// TIA Portal V17 export
// export: Created 2023-02-25T14:39:28.1459249Z, ExportSetting WithDefaults, DisplayName Totally Integrated Automation Portal, DisplayVersion V17, DisplayName TIA Portal Openness, DisplayVersion V17, DisplayName TIA Portal Version Control Interface, DisplayVersion V17, DisplayName TIA Portal Test Suite Advanced, DisplayVersion V17, DisplayName STEP 7 Professional, DisplayVersion V17, DisplayName SIMATIC Energy Suite, DisplayVersion V17, DisplayName STEP 7 Safety, DisplayVersion V17, DisplayName WinCC Professional, DisplayVersion V17
FUNCTION_BLOCK "HW_MotorControle"   // FB1, LAD
{ S7_Optimized_Access := 'TRUE' }
VERSION : 0.1
// stored: AutoNumber true, IsIECCheckEnabled false, IsRetainMemResEnabled false, MemoryReserve 100, SetENOAutomatically false, UDAEnableTagReadback false
   VAR_INPUT
      inConveyor : "stt_Motor";
      FirstScan : Bool;
   END_VAR
   VAR_OUTPUT
      Conveyor : Real;
   END_VAR
   VAR
      S1 : Bool;
      S2 : Bool;
      S3 : Bool;
      S4 : Bool;
      S5 : Bool;
      t1 : Bool;
      t2 : Bool;
      speedLeft : Real;
      IEC_Timer_0_Instance { ExternalAccessible := 'False'; ExternalVisible := 'False'; ExternalWritable := 'False'} : TON_TIME;
      IEC_Timer_0_Instance_1 { ExternalAccessible := 'False'; ExternalVisible := 'False'; ExternalWritable := 'False'} : TON_TIME;
   END_VAR
BEGIN

REGION Network 1: Step 2-1
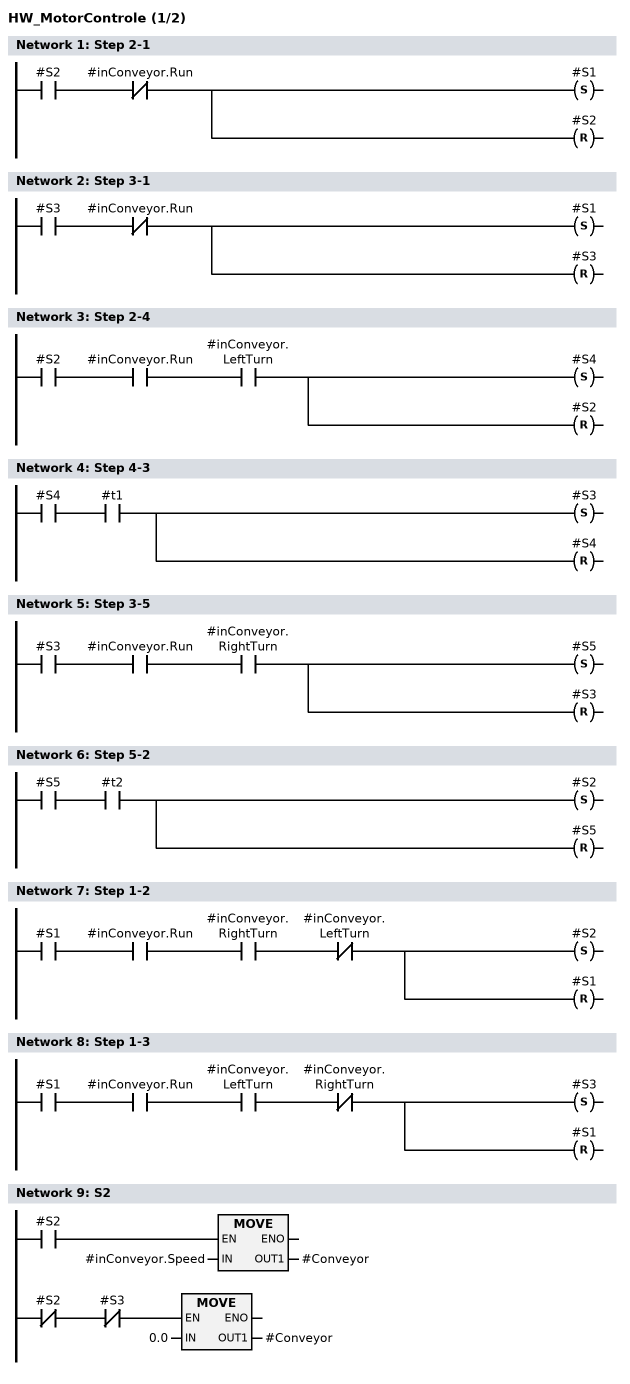
   RUNG wire#powerrail
      Contact( #S2 )
      I_Contact( #inConveyor.Run )
      wire#w1
      S_Coil( #S1 )
   END_RUNG
   RUNG wire#w1
      R_Coil( #S2 )
   END_RUNG
   // the same network as SCL:
   IF #S2 AND NOT #inConveyor.Run THEN
       #S1 := TRUE;
       #S2 := FALSE;
   END_IF;
END_REGION

REGION Network 2: Step 3-1
   RUNG wire#powerrail
      Contact( #S3 )
      I_Contact( #inConveyor.Run )
      wire#w1
      S_Coil( #S1 )
   END_RUNG
   RUNG wire#w1
      R_Coil( #S3 )
   END_RUNG
   // the same network as SCL:
   IF #S3 AND NOT #inConveyor.Run THEN
       #S1 := TRUE;
       #S3 := FALSE;
   END_IF;
END_REGION

REGION Network 3: Step 2-4
   RUNG wire#powerrail
      Contact( #S2 )
      Contact( #inConveyor.Run )
      Contact( #inConveyor.LeftTurn )
      wire#w1
      S_Coil( #S4 )
   END_RUNG
   RUNG wire#w1
      R_Coil( #S2 )
   END_RUNG
   // the same network as SCL:
   IF #S2 AND #inConveyor.Run AND #inConveyor.LeftTurn THEN
       #S4 := TRUE;
       #S2 := FALSE;
   END_IF;
END_REGION

REGION Network 4: Step 4-3
   RUNG wire#powerrail
      Contact( #S4 )
      Contact( #t1 )
      wire#w1
      S_Coil( #S3 )
   END_RUNG
   RUNG wire#w1
      R_Coil( #S4 )
   END_RUNG
   // the same network as SCL:
   IF #S4 AND #t1 THEN
       #S3 := TRUE;
       #S4 := FALSE;
   END_IF;
END_REGION

REGION Network 5: Step 3-5
   RUNG wire#powerrail
      Contact( #S3 )
      Contact( #inConveyor.Run )
      Contact( #inConveyor.RightTurn )
      wire#w1
      S_Coil( #S5 )
   END_RUNG
   RUNG wire#w1
      R_Coil( #S3 )
   END_RUNG
   // the same network as SCL:
   IF #S3 AND #inConveyor.Run AND #inConveyor.RightTurn THEN
       #S5 := TRUE;
       #S3 := FALSE;
   END_IF;
END_REGION

REGION Network 6: Step 5-2
   RUNG wire#powerrail
      Contact( #S5 )
      Contact( #t2 )
      wire#w1
      S_Coil( #S2 )
   END_RUNG
   RUNG wire#w1
      R_Coil( #S5 )
   END_RUNG
   // the same network as SCL:
   IF #S5 AND #t2 THEN
       #S2 := TRUE;
       #S5 := FALSE;
   END_IF;
END_REGION

REGION Network 7: Step 1-2
   RUNG wire#powerrail
      Contact( #S1 )
      Contact( #inConveyor.Run )
      Contact( #inConveyor.RightTurn )
      I_Contact( #inConveyor.LeftTurn )
      wire#w1
      S_Coil( #S2 )
   END_RUNG
   RUNG wire#w1
      R_Coil( #S1 )
   END_RUNG
   // the same network as SCL:
   IF #S1 AND #inConveyor.Run AND #inConveyor.RightTurn AND NOT #inConveyor.LeftTurn THEN
       #S2 := TRUE;
       #S1 := FALSE;
   END_IF;
END_REGION

REGION Network 8: Step 1-3
   RUNG wire#powerrail
      Contact( #S1 )
      Contact( #inConveyor.Run )
      Contact( #inConveyor.LeftTurn )
      I_Contact( #inConveyor.RightTurn )
      wire#w1
      S_Coil( #S3 )
   END_RUNG
   RUNG wire#w1
      R_Coil( #S1 )
   END_RUNG
   // the same network as SCL:
   IF #S1 AND #inConveyor.Run AND #inConveyor.LeftTurn AND NOT #inConveyor.RightTurn THEN
       #S3 := TRUE;
       #S1 := FALSE;
   END_IF;
END_REGION

REGION Network 9: S2
   RUNG wire#powerrail
      Contact( #S2 )
      Move(in := #inConveyor.Speed, out1 => #Conveyor)
   END_RUNG
   RUNG wire#powerrail
      I_Contact( #S2 )
      I_Contact( #S3 )
      Move(in := 0.0, out1 => #Conveyor)
   END_RUNG
   // the same network as SCL:
   IF #S2 THEN #Conveyor := #inConveyor.Speed; END_IF;
   IF NOT #S2 AND NOT #S3 THEN #Conveyor := 0.0; END_IF;
END_REGION

REGION Network 10: S3
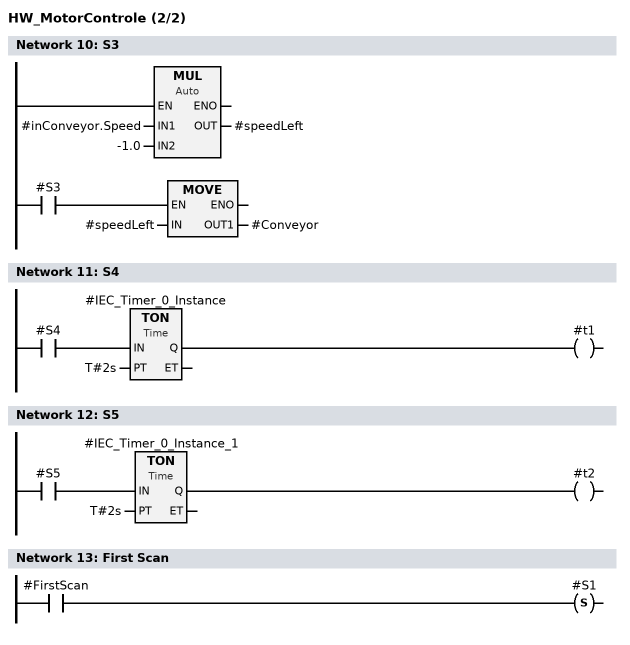
   RUNG wire#powerrail
      Mul(in1 := #inConveyor.Speed, in2 := -1.0, out => #speedLeft)
   END_RUNG
   RUNG wire#powerrail
      Contact( #S3 )
      Move(in := #speedLeft, out1 => #Conveyor)
   END_RUNG
   // the same network as SCL:
   #speedLeft := #inConveyor.Speed * (-1.0);
   IF #S3 THEN #Conveyor := #speedLeft; END_IF;
END_REGION

REGION Network 11: S4
   RUNG wire#powerrail
      Contact( #S4 )
      { S7_Templates := "time_type := Time" } #IEC_Timer_0_Instance.TON(pt := T#2s, et =>)
      Coil( #t1 )
   END_RUNG
   // the same network as SCL:
   #IEC_Timer_0_Instance(IN := #S4, PT := T#2s);   // TON
   #t1 := #IEC_Timer_0_Instance.Q;
END_REGION

REGION Network 12: S5
   RUNG wire#powerrail
      Contact( #S5 )
      { S7_Templates := "time_type := Time" } #IEC_Timer_0_Instance_1.TON(pt := T#2s, et =>)
      Coil( #t2 )
   END_RUNG
   // the same network as SCL:
   #IEC_Timer_0_Instance_1(IN := #S5, PT := T#2s);   // TON
   #t2 := #IEC_Timer_0_Instance_1.Q;
END_REGION

REGION Network 13: First Scan
   RUNG wire#powerrail
      Contact( #FirstScan )
      S_Coil( #S1 )
   END_RUNG
   // the same network as SCL:
   IF #FirstScan THEN #S1 := TRUE; END_IF;
END_REGION
END_FUNCTION_BLOCK
